(* Logix 5000 project; controller Joltek_RA_5069PLC002 vendor 1 type 14 code 226 rev 34.15; software revision 34.04 *)

TASK MainTask (continuous, watchdog 500 ms) : MainProgram
TASK SafetyTask (periodic, rate 20 ms, priority 10, watchdog 20 ms, safety) : SafetyProgram

MODULES
   Local : vendor 1 type 14 code 226 (5069 0, rev 34.15)
      Joltek_SW001 : vendor 1 type 12 code 231 (Ethernet 192.168.1.70, rev 13.8, Output RPI 1000 ms)
END_MODULES

TYPE UDT_ErrorDataLog :
STRUCT
   Time : UDT_Timestamp;
   DINTlog : DINT[10];
   REALlog : REAL[10];
END_STRUCT
END_TYPE

TYPE UDT_Line :
STRUCT
   Filler : UDT_Machine;
   Capper : UDT_Machine;
   Labeler : UDT_Machine;
   CasePAcker : UDT_Machine;
END_STRUCT
END_TYPE

TYPE UDT_Machine :
STRUCT
   Status : INT;
   Running : TIMER;
   Running_B : BOOL;
   CustomData : DINT[10];
   CustomREALData : REAL[10];
   Faulted : DINT;
END_STRUCT
END_TYPE

TYPE UDT_MachineData :
STRUCT
   CurrHourProdMade : INT;
   Prev120ShiftProdMade : INT[120];
   Last8HoursProdMade : INT[8];
   ResettableProdMade : DINT;
END_STRUCT
END_TYPE

TYPE UDT_Timestamp :
STRUCT
   Year : DINT;
   Month : DINT;
   Day : DINT;
   Hour : DINT;
   Minute : DINT;
   Second : DINT;
END_STRUCT
END_TYPE

TYPE UDT_TimestampedData :
STRUCT
   Hour : INT;
   Minute : INT;
   Second : INT;
   Data1 : DINT;
   Data2 : DINT;
   Data3 : DINT;
   Data_BOOL : BOOL[32];
   Data_REAL : REAL[5];
END_STRUCT
END_TYPE

VAR_GLOBAL   (* controller tags *)
   HMI_BOOL1 : BOOL[128] := ([0] := 1);
        [2]   // Filler - HMI | Station 1 Filling
        [3]   // Filler - HMI | Station 2 Filling
   HMI_INT : INT[100] := ([0] := 1, [1] := 96, [2] := 14, [3] := 16652, [4] := 88, [10] := 3, [11] := 40, [12] := 9134, [14] := 9, [20] := 2, [23] := 2056, [30] := 2, [31] := 9850, [32] := 70, [33] := 4100, [40] := 3, [41] := 9, [42] := 45, [50] := 4, [51] := 22, [52] := 7, [56] := 22, [57] := 7, [61] := 22, [62] := 7, [67] := 22, [68] := 7);
        [50].0   // Line - HIM | Start Permissive
        [3].13   // Filler HMI - Start Command
        [50].1   // Line - HIM | Start Command
        [50].2   // Line - HIM | Stop Permissive
        [50].3   // Line - HIM | Stop Command
        [23].1   // Labeler - Start Permissive
        [50].5   // Line - HIM | Fault Reset Command
        [23].3   // Labeler - Stop Permissive
        [23].4   // Labeler - HMI Stop Command
        [23].5   // Labeler - HMI Faulted Status
        [23].6   // Labeler - HMI Fault Reset Command
        [33].0   // Case Packer - HMI | Case Folding in Progress
        [33].1   // Case Packer - HMI | Case Gluing in Progress
        [33].10   // Case Packer - HMI | Start Permissive
        [33].11   // Case Packer - HMI | Start Command
        [33].12   // Case Packer - HMI | Stop Permissive
        [33].13   // Case Packer - HMI | Stop Command
        [33].15   // Case Packer - HMI | Clear Fault Command
        [41].0   // Palletizer - HMI | Currently Palletizing
        [14].6   // Capper - HMI | Fault Reset Command
        [41].1   // Palletizer - HMI | Start Permissive
        [23].2   // Labeler - HMI Start Command
        [23].0   // Labeler - Labeling in Process
        [3].12   // Filler - Start Permissive
        [41].2   // Palletizer - HMI | Start Command
        [14].2   // Capper - HMI | Start Command
        [41].7   // Palletizer - HMI | Clear Pallet Command
        [14].4   // Capper - HMI | Stop Command
        [4].2   // Filler - HMI | Add Bottles to Infeed
        [4].3   // Filler - HMI | Add Bottles to Infeed Permissive
        [4].4   // Overall - HMI | Count Reset Permissive
        [4].5   // Overall - HMI | Count Reset
        [4].7   // Overall - HMI | All Data Reset
        [4].6   // Overall - HMI | All Data Reset Permissive
   HMI_REAL : REAL[100] := ([0] := 46.01, [1] := 36.01, [2] := 100.0, [4] := 100.0, [7] := 100.0);
   LabelerNumberOfStops : COUNTER := (ACC := 16, DN := 1);
   LabelerStop_Data1ARR : DINT[100] := ([0] := 212, [1] := 209);
   LabelerStop_Data1CTR : CONTROL := (LEN := 100, POS := 2);
   LabelerStop_Data2CTR : CONTROL := (LEN := 100, POS := 5);
   LabelerStop_Hour : DINT := 10;
   LabelerStop_HourARR : DINT[100] := ([0] := 11, [1] := 11);
   LabelerStop_HourCTR : CONTROL := (LEN := 100, POS := 2);
   LabelerStop_MinCTR : CONTROL := (LEN := 100, POS := 2);
   LabelerStop_Minute : DINT := 2;
   LabelerStop_MinuteARR : DINT[100] := ([0] := 43, [1] := 43);
   LabelerStop_ONS : BOOL;
   LabelerStop_SecCTR : CONTROL := (LEN := 100, POS := 2);
   LabelerStop_Second : DINT := 37;
   LabelerStop_SecondARR : DINT[100] := ([0] := 11, [1] := 30);
   LabelerStopData : UDT_TimestampedData[100] := ([0].Hour := 12, [0].Minute := 24, [0].Second := 59, [0].Data1 := 193, [0].Data2 := 40, [0].Data3 := 6, [1].Hour := 12, [1].Minute := 25, [1].Second := 27, [1].Data1 := 188, [1].Data2 := 40, [1].Data3 := 5, [2].Hour := 22, [2].Minute := 24, [2].Second := 31, [2].Data1 := 188, [2].Data2 := 40, [2].Data3 := 5, [3].Hour := 10, [3].Second := 20, [3].Data1 := 249, [3].Data2 := 40, [3].Data3 := 2, [4].Hour := 10, [4].Minute := 2, [4].Second := 37, [4].Data1 := 246, [4].Data2 := 40, [4].Data3 := 5);
   LabelerStopDataONE : UDT_TimestampedData := (Hour := 10, Minute := 2, Second := 37, Data1 := 246, Data2 := 40, Data3 := 5);
   LabelerStops : COUNTER := (ACC := 3, CU := 1, DN := 1);
   Line1 : UDT_Line;
   Line34Pump3Motor342DischargeOfTank23_Sig : DINT;
   Line45Pump3MTR345InfeedRawIngredientFlou : DINT;
   Line6Pump1DischargeOfTank3 : DINT;
   Sys_DINT : DINT[100] := ([0] := 3, [1] := 1796, [2] := 6546, [3] := 49412, [4] := 96, [5] := 4601, [6] := 3601, [7] := 1, [8] := 1, [9] := 1, [10] := 1, [11] := 1, [12] := 1, [13] := 1, [14] := 1, [15] := 1, [16] := 1, [17] := 1, [18] := 1, [19] := 1, [20] := 1, [21] := 1, [22] := 1, [23] := 1, [24] := 1, [25] := 1, [26] := 1, [27] := 1, [28] := 1, [29] := 1, [30] := 1, [31] := 1, [32] := 1, [33] := 1, [34] := 1, [35] := 1, [36] := 1, [39] := 14, [40] := 52, [41] := 10000, [42] := 40, [43] := 9134, [44] := 516, [48] := 4, [49] := 9850, [51] := 205100, [53] := 70, [54] := 1, [55] := 20, [56] := 10000, [57] := 45, [58] := 22, [59] := 22, [60] := 7, [64] := 25, [65] := 22, [66] := 7);
        [0]   // Line 1 Motor 324 of the Conveyor 23 Discharge Pump 4-20mA Signal
        [40].4   // Capper - Start Capping Process
        [54].0   // Case Packer - Infeed Labeled Bottles Empty
        [1]   // Line 2 Motor 32334 of the Conveyor 2233 Discharge Pump 0-20mA Signal SCALED
        [55].1   // Palletizer - Stop
        [48].4   // Case Packer - Case Filling Station
        [3].4   // Filler - Alarm | Infeed Empty Bottle Conveyor Empty
        [48].5   // Case Packer - Gluing Station Case in Place
        [40].0   // Capper - Start
        [3].7   // Filler - Alarm | Discharge Filled Bottle Conveyor Almost Full
        [48].6   // Case Packer - Case Filled Ready
        [40].5   // Capper Discharge Conveyor Full
        [54].1   // Case Packer - Infeed Labeled Bottles Low
        [55].2   // Palletizer - Running
        [40].1   // Capper - Stop
        [3].6   // Filler - Alarm | Discharge Filled Bottle Conveyor Full
        [40].6   // Capper Discharge Conveyor Almost Full
        [40].2   // Capper - Running
        [3].2   // Filler - Running
        [44].0   // Labeler - Start
        [44].1   // Labeler - Stop
        [44].10   // Labeler - Unwind Station Almost Empty
        [44].2   // Labeler - Running
        [44].3   // Labeler - Faulted
        [44].5   // Labeler - Labeled Bottle Conveyor Full
        [44].6   // Labeler - Labeled Bottle Conveyor Almost Full
        [44].7   // Labeler - Capped Bottle Conveyor Empty
        [44].8   // Labeler - Capped Bottle Conveyor Almost Empty
        [44].9   // Labeler - Unwind Station Empty
        [46]   // Labeled Bollte Conveyor Count
        [48].0   // Case Packer - Start
        [48].7   // Case Packer - Gluing Station Case Start
        [3].3   // Filler - Faulted
        [55].3   // Palletizer - Faulted
        [54].2   // Case Packer - Cases Empty
        [54].3   // Case Packer - Cases Low
        [40].7   // Capper Infeed Conveyor Empty
        [3].5   // Filler - Alarm | Infeed Empty Bottle Conveyor Low
        [40].8   // Capper Infeed Conveyor Almost Empty
        [49]   // Case Packer - Empty Case Count
        [54].4   // Case Packer - Glue Tank Empty
        [43]   // Capper - Caps available in the hopper
        [55].4   // Palletizer - Case Placed by Robot
        [48].1   // Case Packer - Stop
        [4]   // Filler - Infeed Empty Bottle Count
        [48].2   // Case Packer - Running
        [51]   // Case Packer - Glue Station Level (10,000)
        [54].5   // Case Packer - Glue Tank Low
        [54].6   // Case Packer - Discharge Conveyor Full
        [48].3   // Case Packer - Faulted
        [54].7   // Case Packer - Discharge Conveyor Almost Full
        [40].3   // Capper - Faulted
        [3].1   // Filler - Stop
        [39]   // Filled Bottle Conveyor Count
        [3].12   // Test - Shift Change
        [3].0   // Filler - Start
        [3].8   // Filler - Bottle Filled
        [55].0   // Palletizer - Start
        [3].19   // Test - Hour Change
        [64]   // Current Hour of the Shift
        [65]   // Current Hour of the Shift
   Sys_FIFO_C : CONTROL[50] := ([0].LEN := 32, [0].POS := 32, [0].DN := 1, [1].LEN := 120, [1].EM := 1, [2].LEN := 120, [2].EM := 1, [3].LEN := 120, [3].EM := 1, [4].LEN := 120, [4].EM := 1, [5].LEN := 120, [5].EM := 1, [6].LEN := 120, [6].POS := 1, [7].DN := 1, [7].EM := 1, [8].DN := 1, [8].EM := 1, [9].DN := 1, [9].EM := 1, [10].DN := 1, [10].EM := 1);
   Sys_Timer : TIMER[100] := ([0].PRE := 50, [0].ACC := 39, [0].EN := 1, [0].TT := 1, [1].PRE := 150, [1].ACC := 139, [1].EN := 1, [1].TT := 1, [2].PRE := 2000, [2].ACC := 2000, [2].EN := 1, [2].DN := 1, [3].PRE := 200, [3].ACC := 18, [3].EN := 1, [3].TT := 1, [4].PRE := 200, [4].ACC := 18, [4].EN := 1, [4].TT := 1, [5].PRE := 1000000, [5].ACC := 8572, [5].EN := 1, [5].TT := 1, [10].PRE := 50, [10].ACC := 18, [10].EN := 1, [10].TT := 1, [11].PRE := 50, [12].PRE := 50, [13].PRE := 100, [14].PRE := 50, [14].ACC := 28, [14].EN := 1, [14].TT := 1);
   System_Date_Time : DINT[7] := ([0] := 2026, [1] := 1, [2] := 15, [3] := 23, [4] := 49, [5] := 38, [6] := 94001);
   Test_Bool : BOOL[64];
   TestBOOL : BOOL;
   TestControl : CONTROL;
   TestCounter : COUNTER;
   TestDINT : DINT;
   TestDINTArray : DINT[10];
   TestINT : INT;
   TestTimer : TIMER;
   TestTimerArr : TIMER[10];
END_VAR

PROGRAM MainProgram   (* main routine MainRoutine *)
VAR
   CapperData : UDT_MachineData := (CurrHourProdMade := 7, Prev120ShiftProdMade[2] := 449, Prev120ShiftProdMade[3] := 480, Prev120ShiftProdMade[4] := 480, Prev120ShiftProdMade[5] := 480, Prev120ShiftProdMade[6] := 480, Prev120ShiftProdMade[7] := 480, Prev120ShiftProdMade[8] := 480, Last8HoursProdMade[1] := 7);
   CasePackerData : UDT_MachineData;
   CurrentPos1 : DINT := 12;
   FillerData : UDT_MachineData := (CurrHourProdMade := 22, Prev120ShiftProdMade[2] := 226, Last8HoursProdMade[1] := 22);
   LabelerData : UDT_MachineData;
   PalletizerData : UDT_MachineData;
   shiftHour : INT := 1;
   Vlad_Test : BOOL[64] := ([0] := 1);
END_VAR

ROUTINE _01_System   (* ladder *)
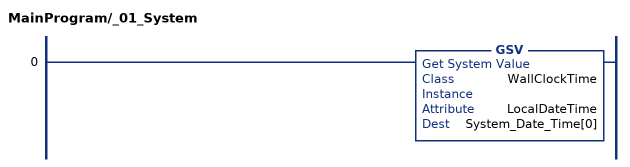
   0: GSV(WallClockTime,,LocalDateTime,System_Date_Time[0]);
END_ROUTINE

ROUTINE _02_Filler   (* ladder *)
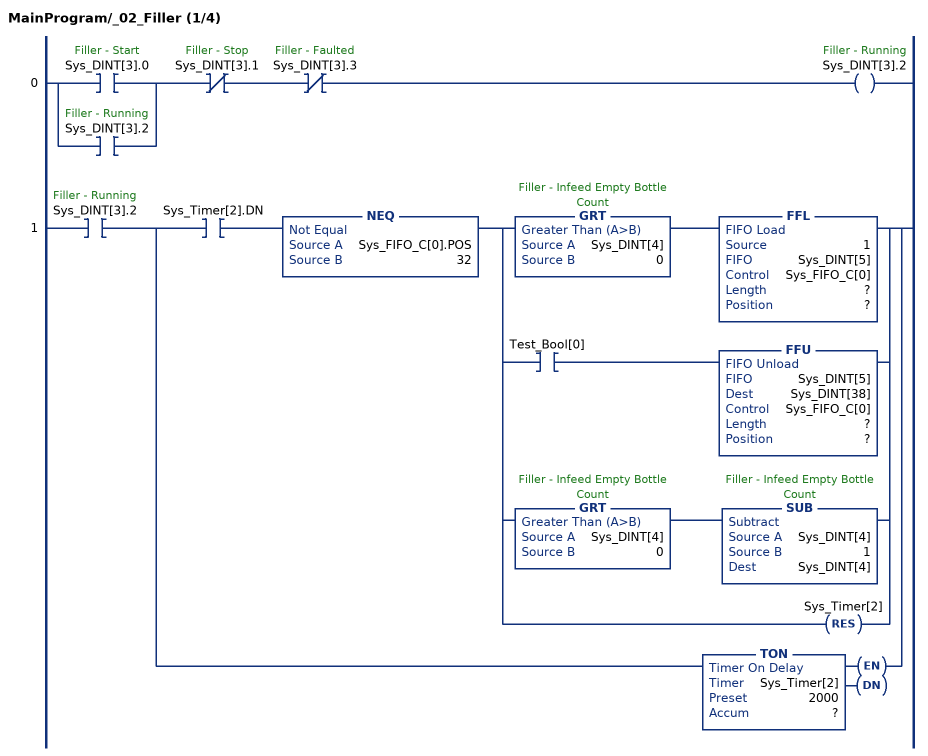
   0: [XIC(Sys_DINT[3].0) ,XIC(Sys_DINT[3].2) ]XIO(Sys_DINT[3].1)XIO(Sys_DINT[3].3)OTE(Sys_DINT[3].2);
   1: XIC(Sys_DINT[3].2)[XIC(Sys_Timer[2].DN) NEQ(Sys_FIFO_C[0].POS,32) [GRT(Sys_DINT[4],0) FFL(1,Sys_DINT[5],Sys_FIFO_C[0],?,?) ,XIC(Test_Bool[0]) FFU(Sys_DINT[5],Sys_DINT[38],Sys_FIFO_C[0],?,?) ,GRT(Sys_DINT[4],0) SUB(Sys_DINT[4],1,Sys_DINT[4]) ,RES(Sys_Timer[2]) ] ,TON(Sys_Timer[2],?,?) ];
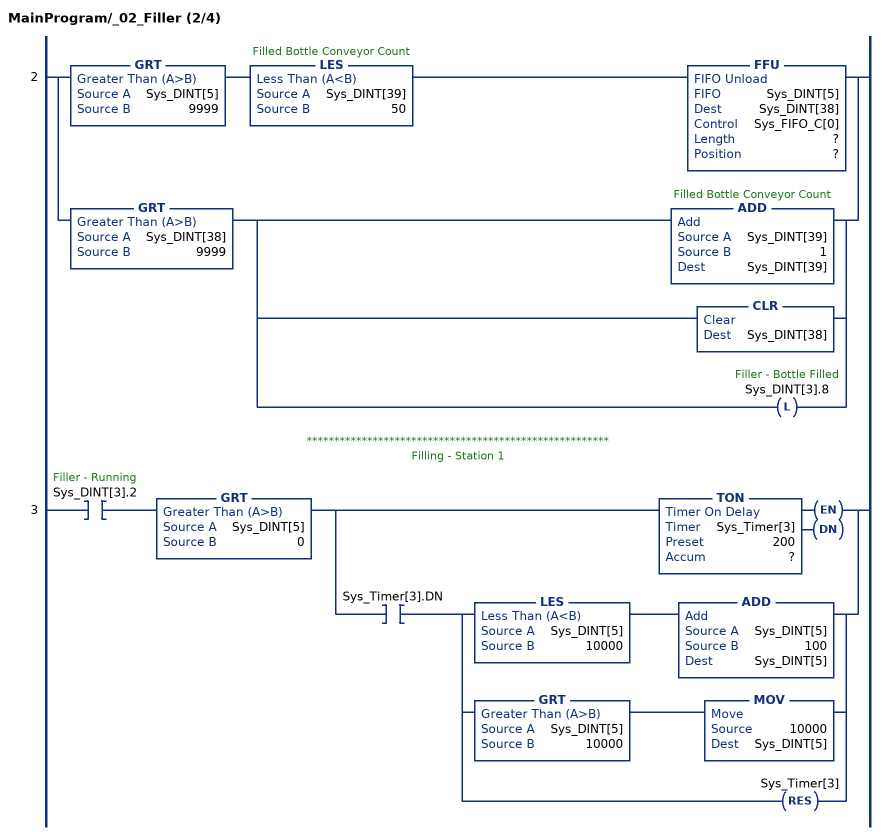
   2: [GRT(Sys_DINT[5],9999) LES(Sys_DINT[39],50) FFU(Sys_DINT[5],Sys_DINT[38],Sys_FIFO_C[0],?,?) ,GRT(Sys_DINT[38],9999) [ADD(Sys_DINT[39],1,Sys_DINT[39]) ,CLR(Sys_DINT[38]) ,OTL(Sys_DINT[3].8) ] ];
   // *******************************************************
   // Filling - Station 1
   3: XIC(Sys_DINT[3].2)GRT(Sys_DINT[5],0)[TON(Sys_Timer[3],?,?) ,XIC(Sys_Timer[3].DN) [LES(Sys_DINT[5],10000) ADD(Sys_DINT[5],100,Sys_DINT[5]) ,GRT(Sys_DINT[5],10000) MOV(10000,Sys_DINT[5]) ,RES(Sys_Timer[3]) ] ];
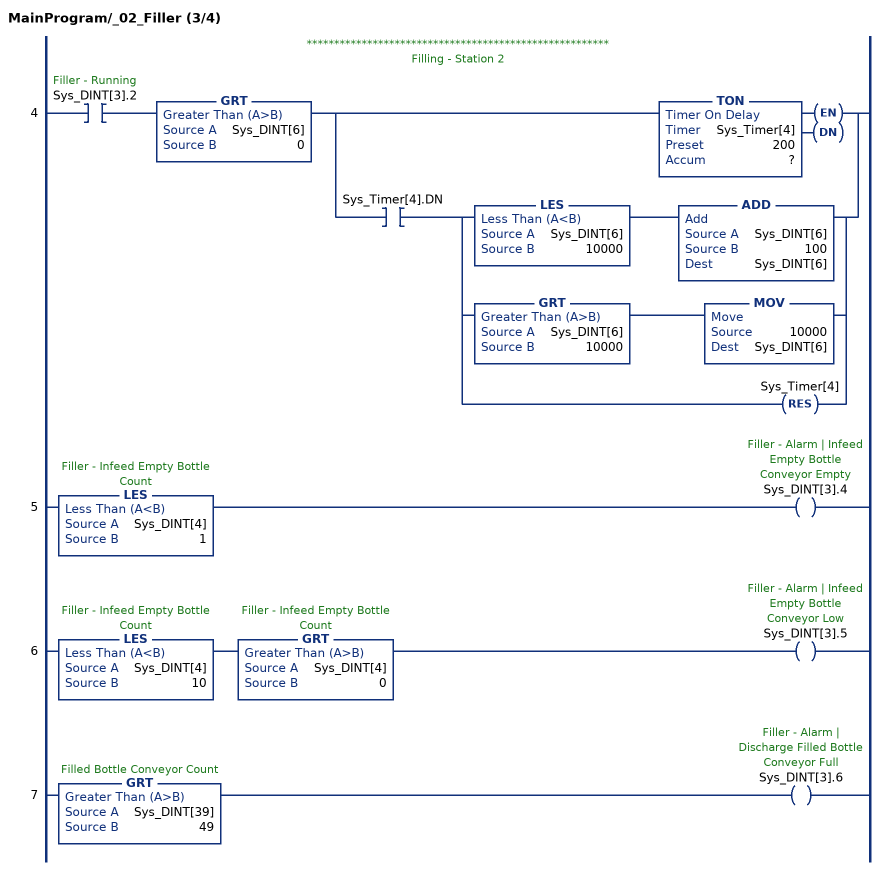
   // *******************************************************
   // Filling - Station 2
   4: XIC(Sys_DINT[3].2)GRT(Sys_DINT[6],0)[TON(Sys_Timer[4],?,?) ,XIC(Sys_Timer[4].DN) [LES(Sys_DINT[6],10000) ADD(Sys_DINT[6],100,Sys_DINT[6]) ,GRT(Sys_DINT[6],10000) MOV(10000,Sys_DINT[6]) ,RES(Sys_Timer[4]) ] ];
   5: LES(Sys_DINT[4],1)OTE(Sys_DINT[3].4);
   6: LES(Sys_DINT[4],10)GRT(Sys_DINT[4],0)OTE(Sys_DINT[3].5);
   7: GRT(Sys_DINT[39],49)OTE(Sys_DINT[3].6);
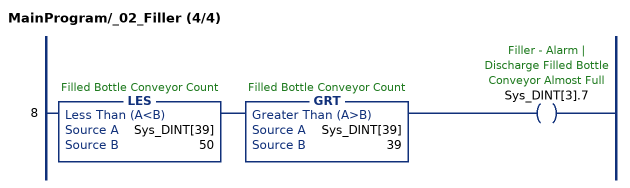
   8: LES(Sys_DINT[39],50)GRT(Sys_DINT[39],39)OTE(Sys_DINT[3].7);
END_ROUTINE

ROUTINE _03_Capper   (* ladder *)
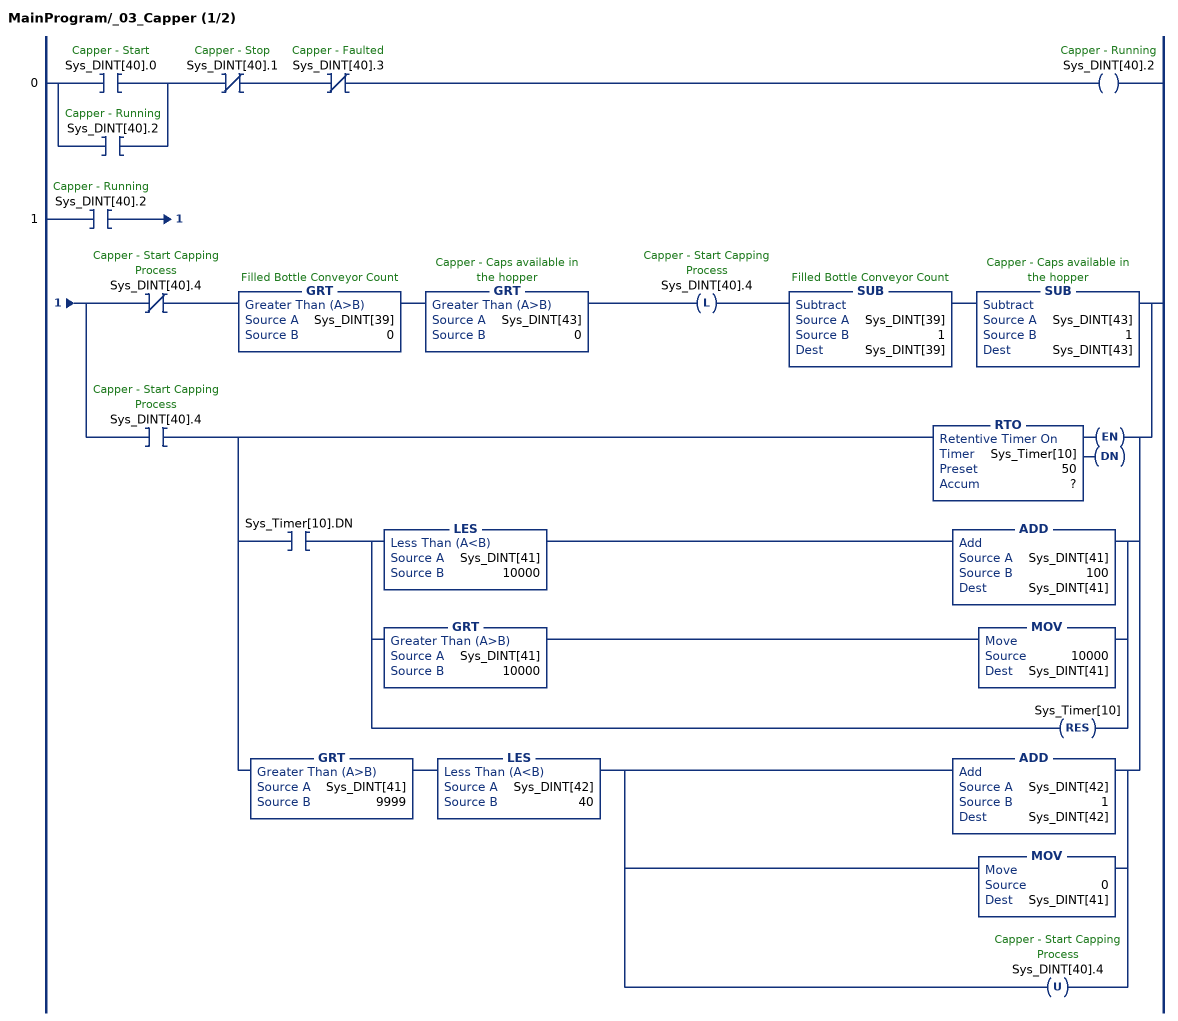
   0: [XIC(Sys_DINT[40].0) ,XIC(Sys_DINT[40].2) ]XIO(Sys_DINT[40].1)XIO(Sys_DINT[40].3)OTE(Sys_DINT[40].2);
   1: XIC(Sys_DINT[40].2)[XIO(Sys_DINT[40].4) GRT(Sys_DINT[39],0) GRT(Sys_DINT[43],0) OTL(Sys_DINT[40].4) SUB(Sys_DINT[39],1,Sys_DINT[39]) SUB(Sys_DINT[43],1,Sys_DINT[43]) ,XIC(Sys_DINT[40].4) [RTO(Sys_Timer[10],?,?) ,XIC(Sys_Timer[10].DN) [LES(Sys_DINT[41],10000) ADD(Sys_DINT[41],100,Sys_DINT[41]) ,GRT(Sys_DINT[41],10000) MOV(10000,Sys_DINT[41]) ,RES(Sys_Timer[10]) ] ,GRT(Sys_DINT[41],9999) LES(Sys_DINT[42],40) [ADD(Sys_DINT[42],1,Sys_DINT[42]) ,MOV(0,Sys_DINT[41]) ,OTU(Sys_DINT[40].4) ] ] ];
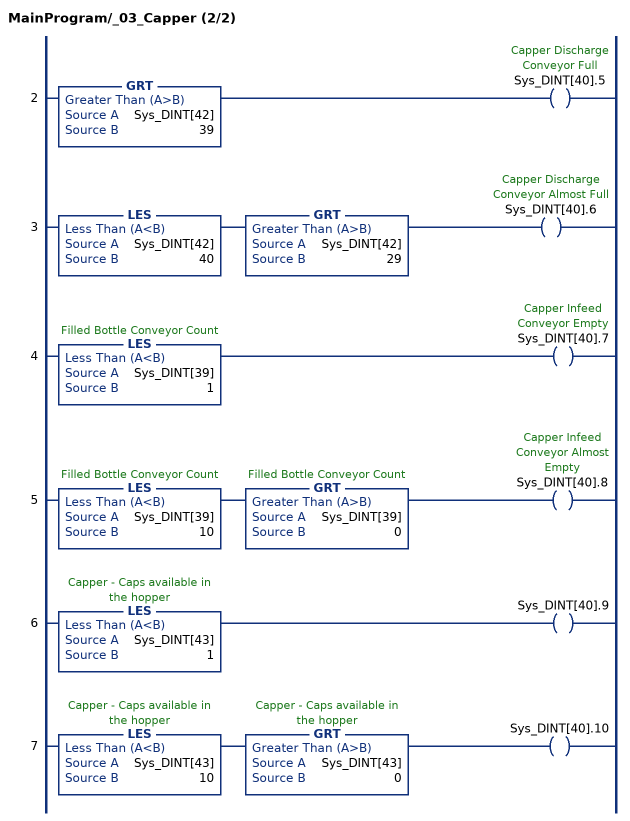
   2: GRT(Sys_DINT[42],39)OTE(Sys_DINT[40].5);
   3: LES(Sys_DINT[42],40)GRT(Sys_DINT[42],29)OTE(Sys_DINT[40].6);
   4: LES(Sys_DINT[39],1)OTE(Sys_DINT[40].7);
   5: LES(Sys_DINT[39],10)GRT(Sys_DINT[39],0)OTE(Sys_DINT[40].8);
   6: LES(Sys_DINT[43],1)OTE(Sys_DINT[40].9);
   7: LES(Sys_DINT[43],10)GRT(Sys_DINT[43],0)OTE(Sys_DINT[40].10);
END_ROUTINE

ROUTINE _04_Labeler   (* ladder *)
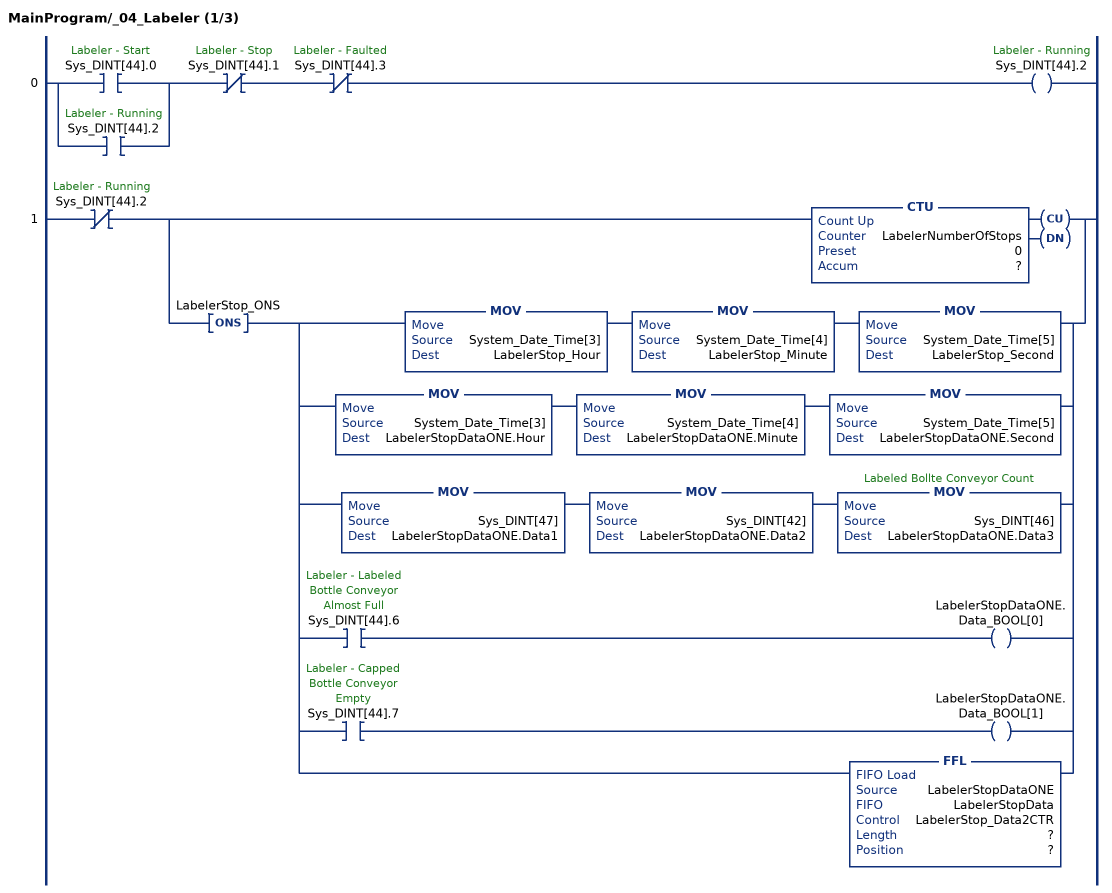
   0: [XIC(Sys_DINT[44].0) ,XIC(Sys_DINT[44].2) ]XIO(Sys_DINT[44].1)XIO(Sys_DINT[44].3)OTE(Sys_DINT[44].2);
   1: XIO(Sys_DINT[44].2)[CTU(LabelerNumberOfStops,?,?) ,ONS(LabelerStop_ONS) [MOV(System_Date_Time[3],LabelerStop_Hour) MOV(System_Date_Time[4],LabelerStop_Minute) MOV(System_Date_Time[5],LabelerStop_Second) ,[MOV(System_Date_Time[3],LabelerStopDataONE.Hour) MOV(System_Date_Time[4],LabelerStopDataONE.Minute) MOV(System_Date_Time[5],LabelerStopDataONE.Second) ,MOV(Sys_DINT[47],LabelerStopDataONE.Data1) MOV(Sys_DINT[42],LabelerStopDataONE.Data2) MOV(Sys_DINT[46],LabelerStopDataONE.Data3) ,[XIC(Sys_DINT[44].6) OTE(LabelerStopDataONE.Data_BOOL[0]) ,XIC(Sys_DINT[44].7) OTE(LabelerStopDataONE.Data_BOOL[1]) ] ,FFL(LabelerStopDataONE,LabelerStopData,LabelerStop_Data2CTR,?,?) ] ] ];
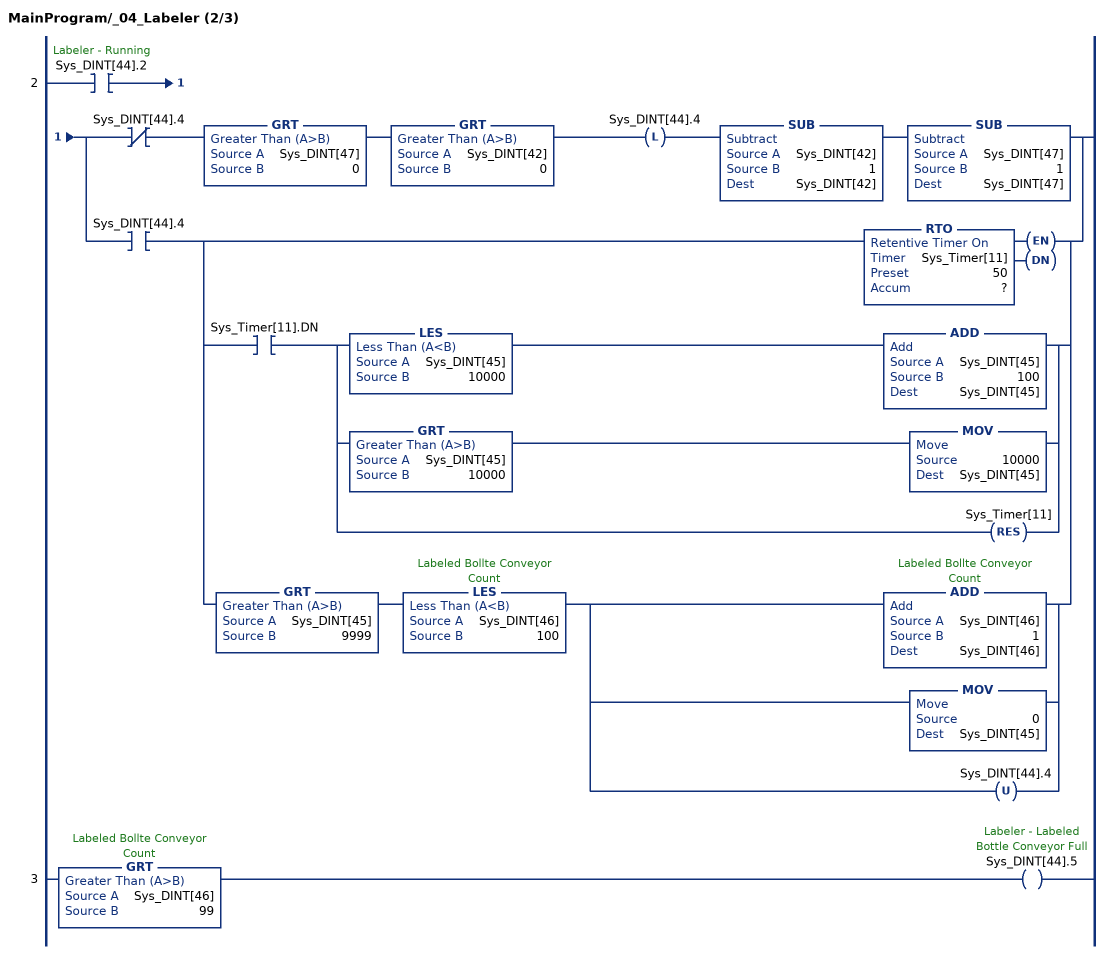
   2: XIC(Sys_DINT[44].2)[XIO(Sys_DINT[44].4) GRT(Sys_DINT[47],0) GRT(Sys_DINT[42],0) OTL(Sys_DINT[44].4) SUB(Sys_DINT[42],1,Sys_DINT[42]) SUB(Sys_DINT[47],1,Sys_DINT[47]) ,XIC(Sys_DINT[44].4) [RTO(Sys_Timer[11],?,?) ,XIC(Sys_Timer[11].DN) [LES(Sys_DINT[45],10000) ADD(Sys_DINT[45],100,Sys_DINT[45]) ,GRT(Sys_DINT[45],10000) MOV(10000,Sys_DINT[45]) ,RES(Sys_Timer[11]) ] ,GRT(Sys_DINT[45],9999) LES(Sys_DINT[46],100) [ADD(Sys_DINT[46],1,Sys_DINT[46]) ,MOV(0,Sys_DINT[45]) ,OTU(Sys_DINT[44].4) ] ] ];
   3: GRT(Sys_DINT[46],99)OTE(Sys_DINT[44].5);
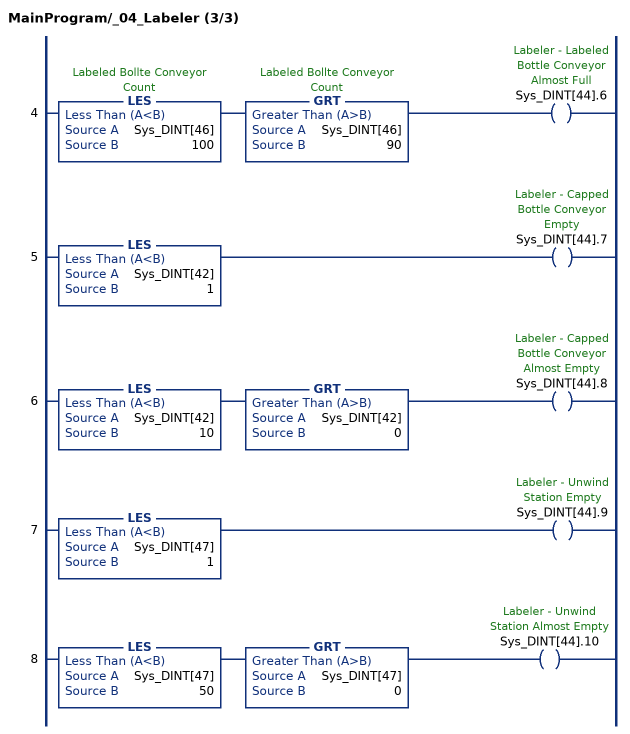
   4: LES(Sys_DINT[46],100)GRT(Sys_DINT[46],90)OTE(Sys_DINT[44].6);
   5: LES(Sys_DINT[42],1)OTE(Sys_DINT[44].7);
   6: LES(Sys_DINT[42],10)GRT(Sys_DINT[42],0)OTE(Sys_DINT[44].8);
   7: LES(Sys_DINT[47],1)OTE(Sys_DINT[44].9);
   8: LES(Sys_DINT[47],50)GRT(Sys_DINT[47],0)OTE(Sys_DINT[44].10);
END_ROUTINE

ROUTINE _05_CasePacker   (* ladder *)
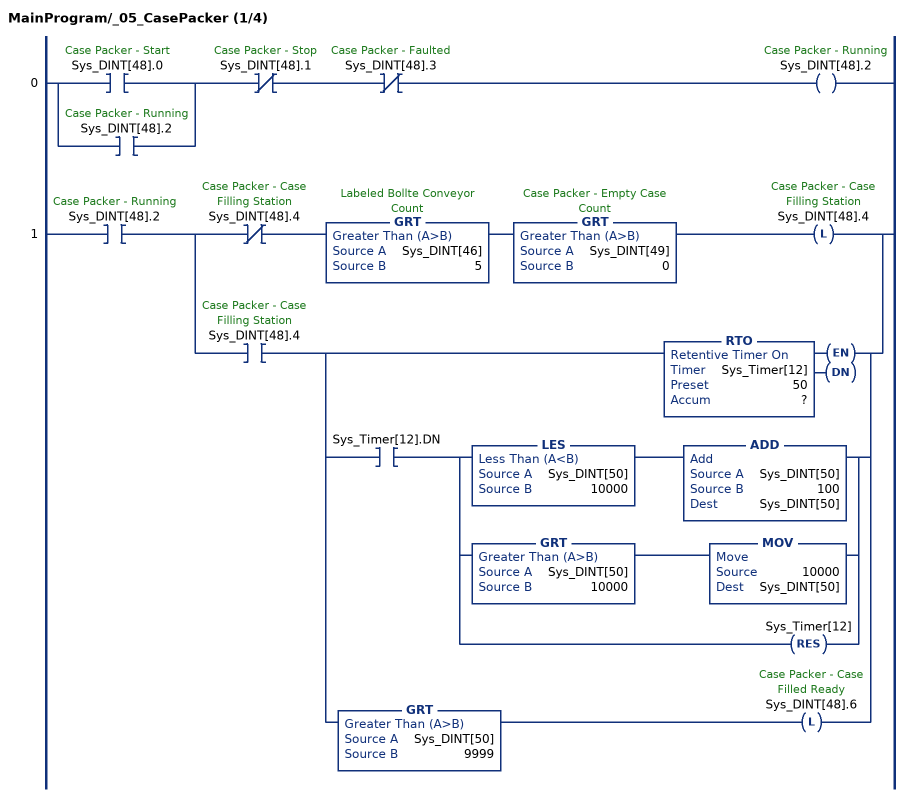
   0: [XIC(Sys_DINT[48].0) ,XIC(Sys_DINT[48].2) ]XIO(Sys_DINT[48].1)XIO(Sys_DINT[48].3)OTE(Sys_DINT[48].2);
   1: XIC(Sys_DINT[48].2)[XIO(Sys_DINT[48].4) GRT(Sys_DINT[46],5) GRT(Sys_DINT[49],0) OTL(Sys_DINT[48].4) ,XIC(Sys_DINT[48].4) [RTO(Sys_Timer[12],?,?) ,XIC(Sys_Timer[12].DN) [LES(Sys_DINT[50],10000) ADD(Sys_DINT[50],100,Sys_DINT[50]) ,GRT(Sys_DINT[50],10000) MOV(10000,Sys_DINT[50]) ,RES(Sys_Timer[12]) ] ,GRT(Sys_DINT[50],9999) OTL(Sys_DINT[48].6) ] ];
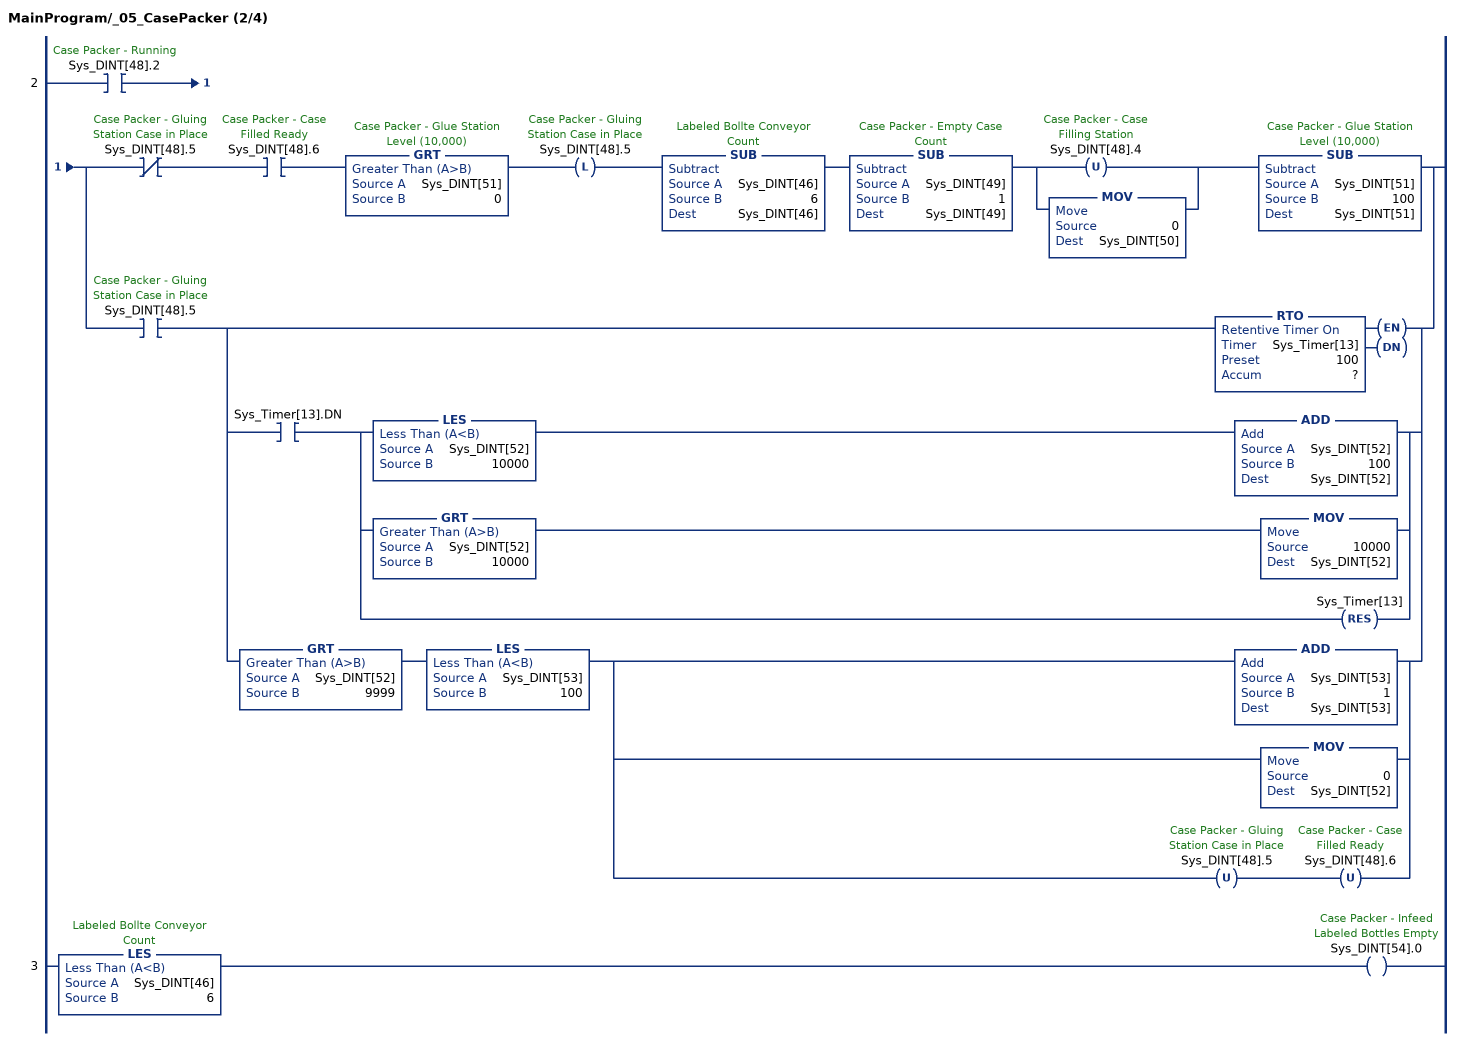
   2: XIC(Sys_DINT[48].2)[XIO(Sys_DINT[48].5) XIC(Sys_DINT[48].6) GRT(Sys_DINT[51],0) OTL(Sys_DINT[48].5) SUB(Sys_DINT[46],6,Sys_DINT[46]) SUB(Sys_DINT[49],1,Sys_DINT[49]) [OTU(Sys_DINT[48].4) ,MOV(0,Sys_DINT[50]) ] SUB(Sys_DINT[51],100,Sys_DINT[51]) ,XIC(Sys_DINT[48].5) [RTO(Sys_Timer[13],?,?) ,XIC(Sys_Timer[13].DN) [LES(Sys_DINT[52],10000) ADD(Sys_DINT[52],100,Sys_DINT[52]) ,GRT(Sys_DINT[52],10000) MOV(10000,Sys_DINT[52]) ,RES(Sys_Timer[13]) ] ,GRT(Sys_DINT[52],9999) LES(Sys_DINT[53],100) [ADD(Sys_DINT[53],1,Sys_DINT[53]) ,MOV(0,Sys_DINT[52]) ,OTU(Sys_DINT[48].5) OTU(Sys_DINT[48].6) ] ] ];
   3: LES(Sys_DINT[46],6)OTE(Sys_DINT[54].0);
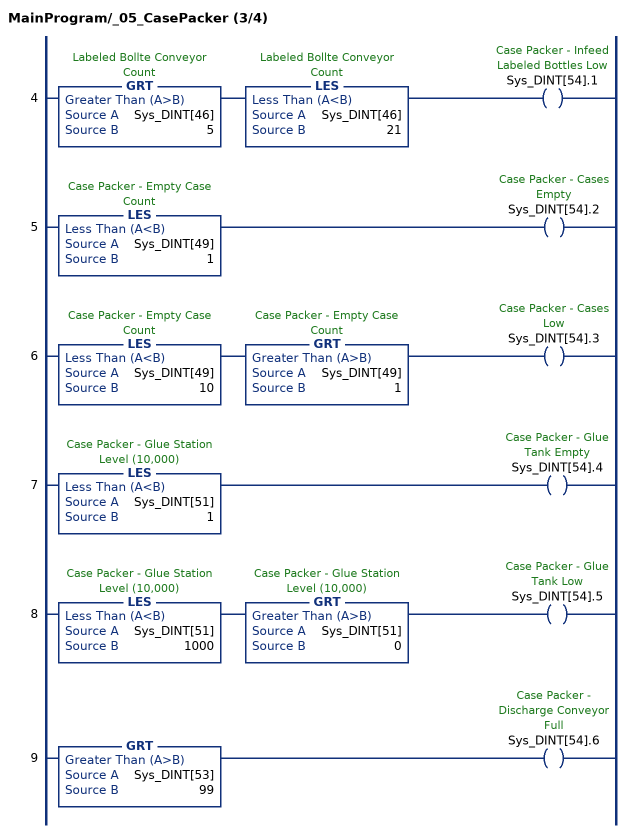
   4: GRT(Sys_DINT[46],5)LES(Sys_DINT[46],21)OTE(Sys_DINT[54].1);
   5: LES(Sys_DINT[49],1)OTE(Sys_DINT[54].2);
   6: LES(Sys_DINT[49],10)GRT(Sys_DINT[49],1)OTE(Sys_DINT[54].3);
   7: LES(Sys_DINT[51],1)OTE(Sys_DINT[54].4);
   8: LES(Sys_DINT[51],1000)GRT(Sys_DINT[51],0)OTE(Sys_DINT[54].5);
   9: GRT(Sys_DINT[53],99)OTE(Sys_DINT[54].6);
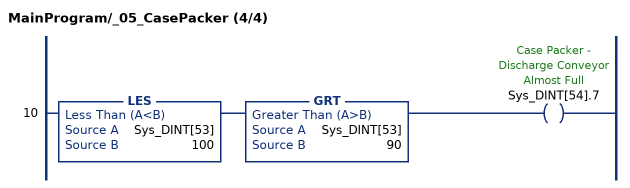
   10: LES(Sys_DINT[53],100)GRT(Sys_DINT[53],90)OTE(Sys_DINT[54].7);
END_ROUTINE

ROUTINE _06_Palletizer   (* ladder *)
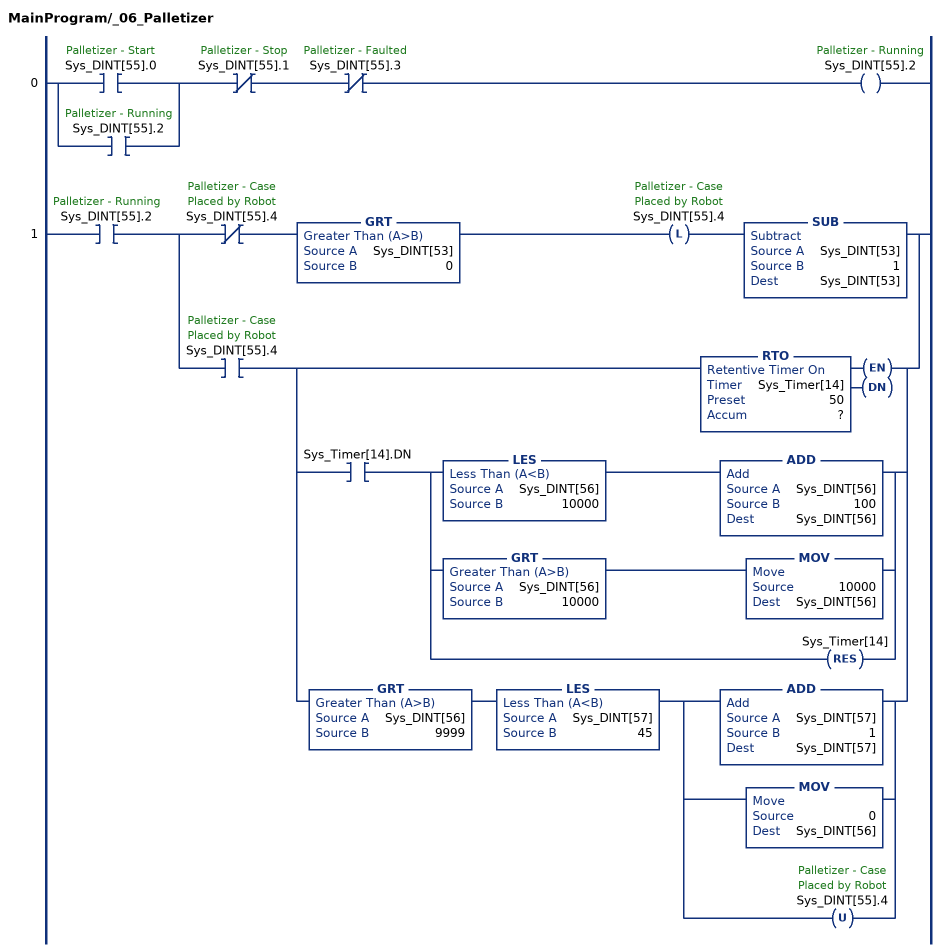
   0: [XIC(Sys_DINT[55].0) ,XIC(Sys_DINT[55].2) ]XIO(Sys_DINT[55].1)XIO(Sys_DINT[55].3)OTE(Sys_DINT[55].2);
   1: XIC(Sys_DINT[55].2)[XIO(Sys_DINT[55].4) GRT(Sys_DINT[53],0) OTL(Sys_DINT[55].4) SUB(Sys_DINT[53],1,Sys_DINT[53]) ,XIC(Sys_DINT[55].4) [RTO(Sys_Timer[14],?,?) ,XIC(Sys_Timer[14].DN) [LES(Sys_DINT[56],10000) ADD(Sys_DINT[56],100,Sys_DINT[56]) ,GRT(Sys_DINT[56],10000) MOV(10000,Sys_DINT[56]) ,RES(Sys_Timer[14]) ] ,GRT(Sys_DINT[56],9999) LES(Sys_DINT[57],45) [ADD(Sys_DINT[57],1,Sys_DINT[57]) ,MOV(0,Sys_DINT[56]) ,OTU(Sys_DINT[55].4) ] ] ];
END_ROUTINE

ROUTINE _50_HMI_Interface   (* ladder *)
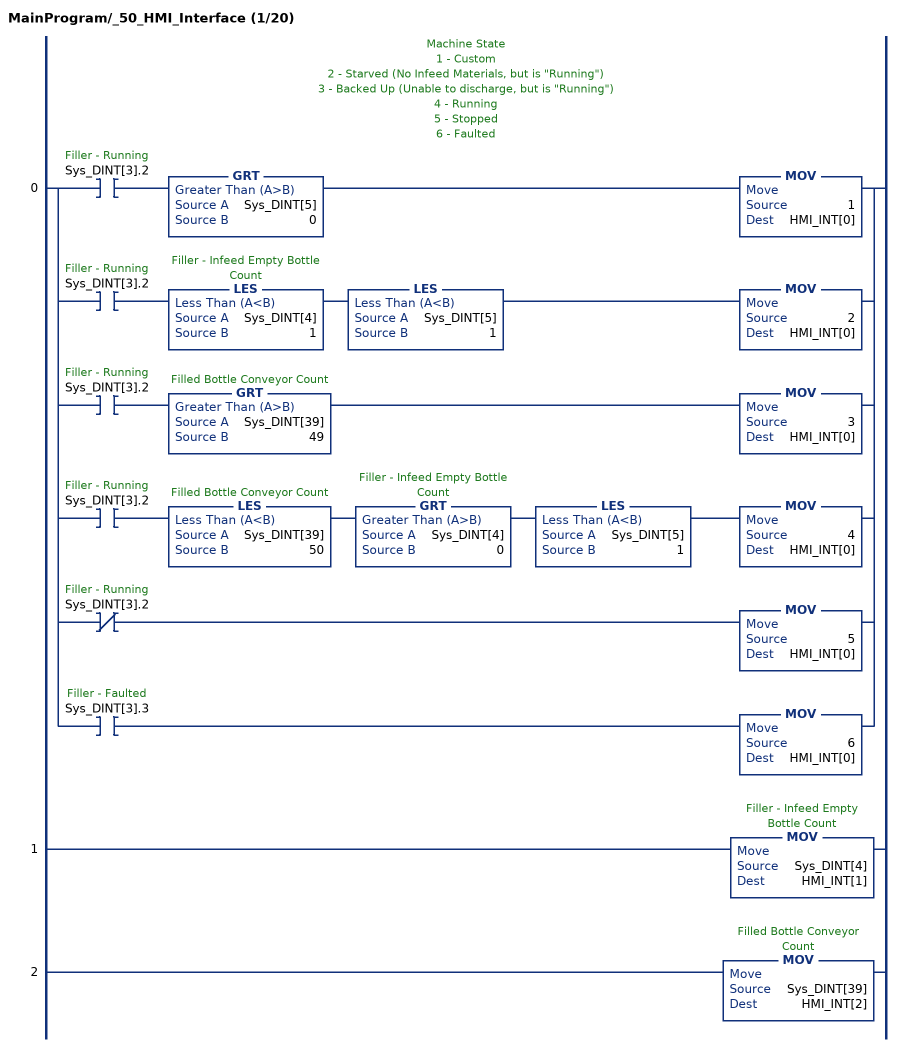
   // Machine State
   // 1 - Custom
   // 2 - Starved (No Infeed Materials, but is "Running")
   // 3 - Backed Up (Unable to discharge, but is "Running")
   // 4 - Running
   // 5 - Stopped
   // 6 - Faulted
   0: [XIC(Sys_DINT[3].2) GRT(Sys_DINT[5],0) MOV(1,HMI_INT[0]) ,XIC(Sys_DINT[3].2) LES(Sys_DINT[4],1) LES(Sys_DINT[5],1) MOV(2,HMI_INT[0]) ,XIC(Sys_DINT[3].2) GRT(Sys_DINT[39],49) MOV(3,HMI_INT[0]) ,XIC(Sys_DINT[3].2) LES(Sys_DINT[39],50) GRT(Sys_DINT[4],0) LES(Sys_DINT[5],1) MOV(4,HMI_INT[0]) ,XIO(Sys_DINT[3].2) MOV(5,HMI_INT[0]) ,XIC(Sys_DINT[3].3) MOV(6,HMI_INT[0]) ];
   1: MOV(Sys_DINT[4],HMI_INT[1]);
   2: MOV(Sys_DINT[39],HMI_INT[2]);
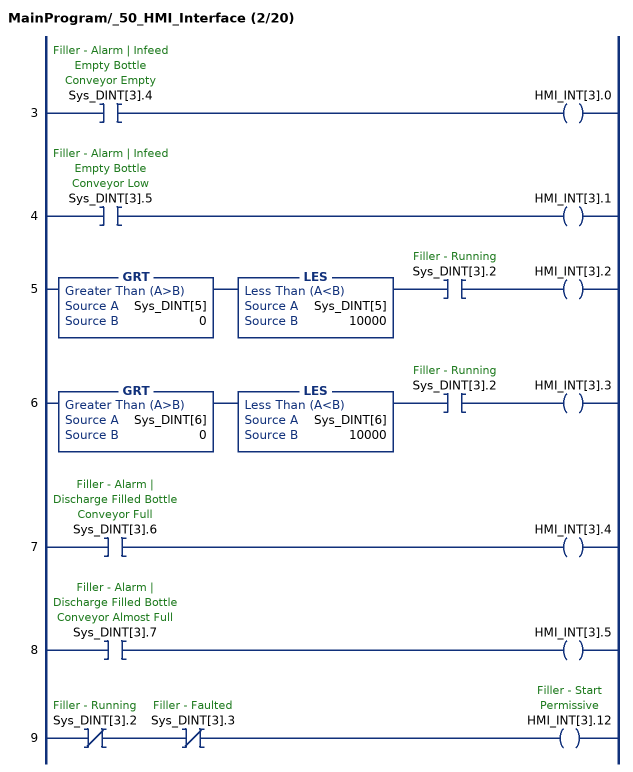
   3: XIC(Sys_DINT[3].4)OTE(HMI_INT[3].0);
   4: XIC(Sys_DINT[3].5)OTE(HMI_INT[3].1);
   5: GRT(Sys_DINT[5],0)LES(Sys_DINT[5],10000)XIC(Sys_DINT[3].2)OTE(HMI_INT[3].2);
   6: GRT(Sys_DINT[6],0)LES(Sys_DINT[6],10000)XIC(Sys_DINT[3].2)OTE(HMI_INT[3].3);
   7: XIC(Sys_DINT[3].6)OTE(HMI_INT[3].4);
   8: XIC(Sys_DINT[3].7)OTE(HMI_INT[3].5);
   9: XIO(Sys_DINT[3].2)XIO(Sys_DINT[3].3)OTE(HMI_INT[3].12);
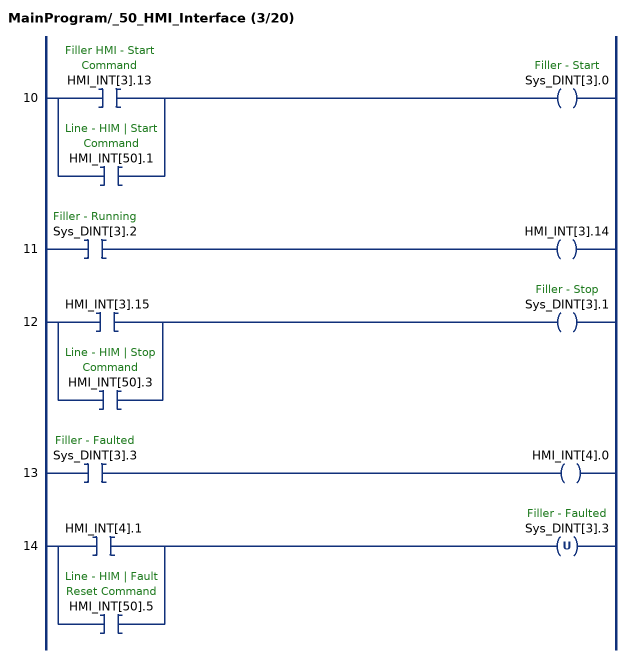
   10: [XIC(HMI_INT[3].13) ,XIC(HMI_INT[50].1) ]OTE(Sys_DINT[3].0);
   11: XIC(Sys_DINT[3].2)OTE(HMI_INT[3].14);
   12: [XIC(HMI_INT[3].15) ,XIC(HMI_INT[50].3) ]OTE(Sys_DINT[3].1);
   13: XIC(Sys_DINT[3].3)OTE(HMI_INT[4].0);
   14: [XIC(HMI_INT[4].1) ,XIC(HMI_INT[50].5) ]OTU(Sys_DINT[3].3);
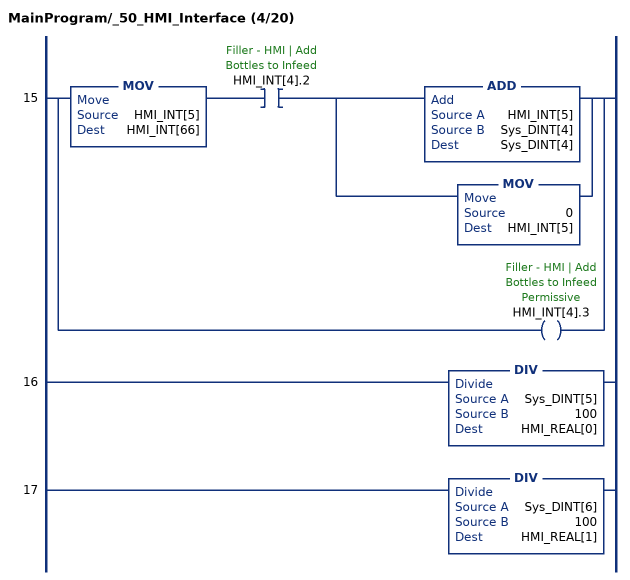
   15: [MOV(HMI_INT[5],HMI_INT[66]) XIC(HMI_INT[4].2) [ADD(HMI_INT[5],Sys_DINT[4],Sys_DINT[4]) ,MOV(0,HMI_INT[5]) ] ,OTE(HMI_INT[4].3) ];
   16: DIV(Sys_DINT[5],100,HMI_REAL[0]);
   17: DIV(Sys_DINT[6],100,HMI_REAL[1]);
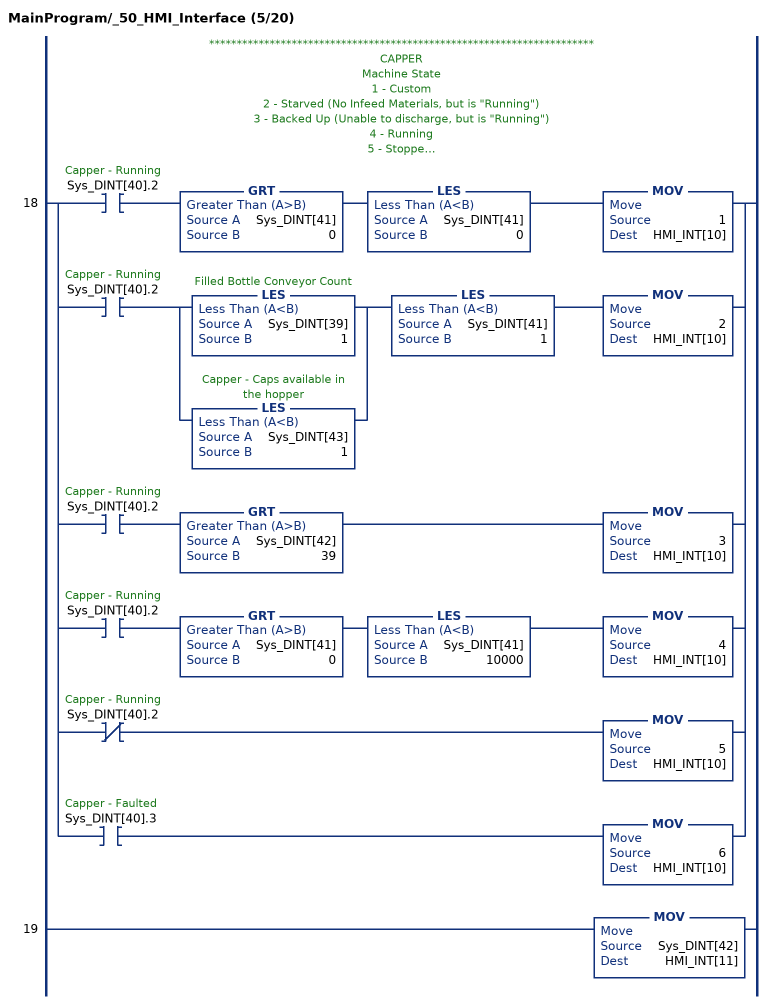
   // **********************************************************************
   // CAPPER
   // Machine State
   // 1 - Custom
   // 2 - Starved (No Infeed Materials, but is "Running")
   // 3 - Backed Up (Unable to discharge, but is "Running")
   // 4 - Running
   // 5 - Stopped
   // 6 - Faulted
   18: [XIC(Sys_DINT[40].2) GRT(Sys_DINT[41],0) LES(Sys_DINT[41],0) MOV(1,HMI_INT[10]) ,XIC(Sys_DINT[40].2) [LES(Sys_DINT[39],1) ,LES(Sys_DINT[43],1) ] LES(Sys_DINT[41],1) MOV(2,HMI_INT[10]) ,XIC(Sys_DINT[40].2) GRT(Sys_DINT[42],39) MOV(3,HMI_INT[10]) ,XIC(Sys_DINT[40].2) GRT(Sys_DINT[41],0) LES(Sys_DINT[41],10000) MOV(4,HMI_INT[10]) ,XIO(Sys_DINT[40].2) MOV(5,HMI_INT[10]) ,XIC(Sys_DINT[40].3) MOV(6,HMI_INT[10]) ];
   19: MOV(Sys_DINT[42],HMI_INT[11]);
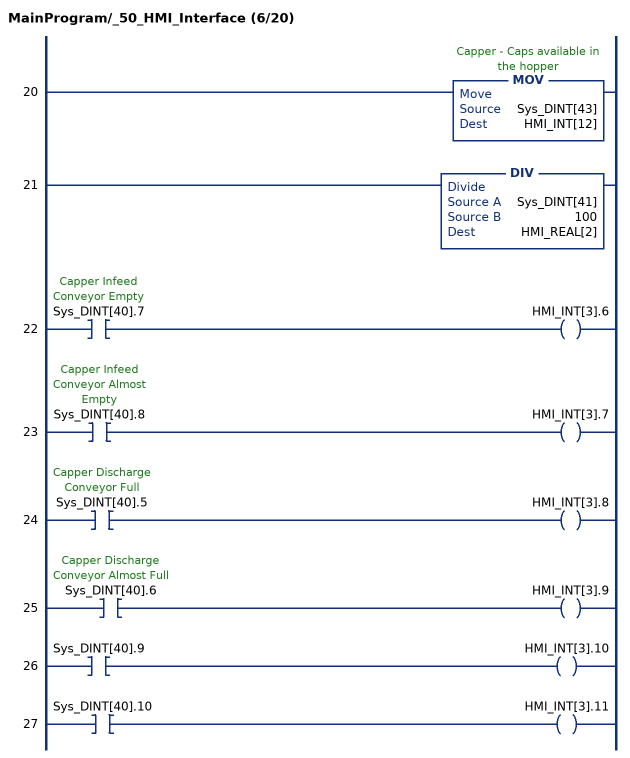
   20: MOV(Sys_DINT[43],HMI_INT[12]);
   21: DIV(Sys_DINT[41],100,HMI_REAL[2]);
   22: XIC(Sys_DINT[40].7)OTE(HMI_INT[3].6);
   23: XIC(Sys_DINT[40].8)OTE(HMI_INT[3].7);
   24: XIC(Sys_DINT[40].5)OTE(HMI_INT[3].8);
   25: XIC(Sys_DINT[40].6)OTE(HMI_INT[3].9);
   26: XIC(Sys_DINT[40].9)OTE(HMI_INT[3].10);
   27: XIC(Sys_DINT[40].10)OTE(HMI_INT[3].11);
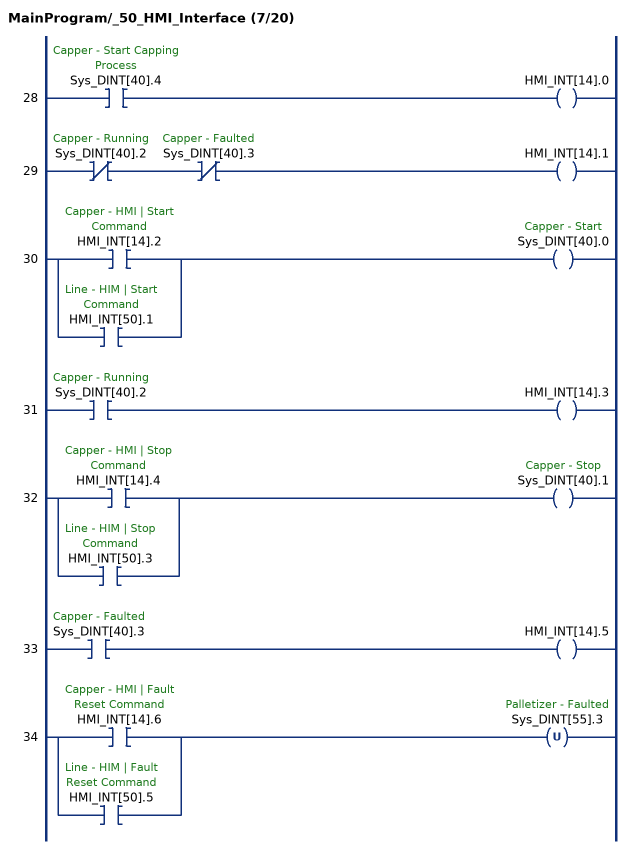
   28: XIC(Sys_DINT[40].4)OTE(HMI_INT[14].0);
   29: XIO(Sys_DINT[40].2)XIO(Sys_DINT[40].3)OTE(HMI_INT[14].1);
   30: [XIC(HMI_INT[14].2) ,XIC(HMI_INT[50].1) ]OTE(Sys_DINT[40].0);
   31: XIC(Sys_DINT[40].2)OTE(HMI_INT[14].3);
   32: [XIC(HMI_INT[14].4) ,XIC(HMI_INT[50].3) ]OTE(Sys_DINT[40].1);
   33: XIC(Sys_DINT[40].3)OTE(HMI_INT[14].5);
   34: [XIC(HMI_INT[14].6) ,XIC(HMI_INT[50].5) ]OTU(Sys_DINT[55].3);
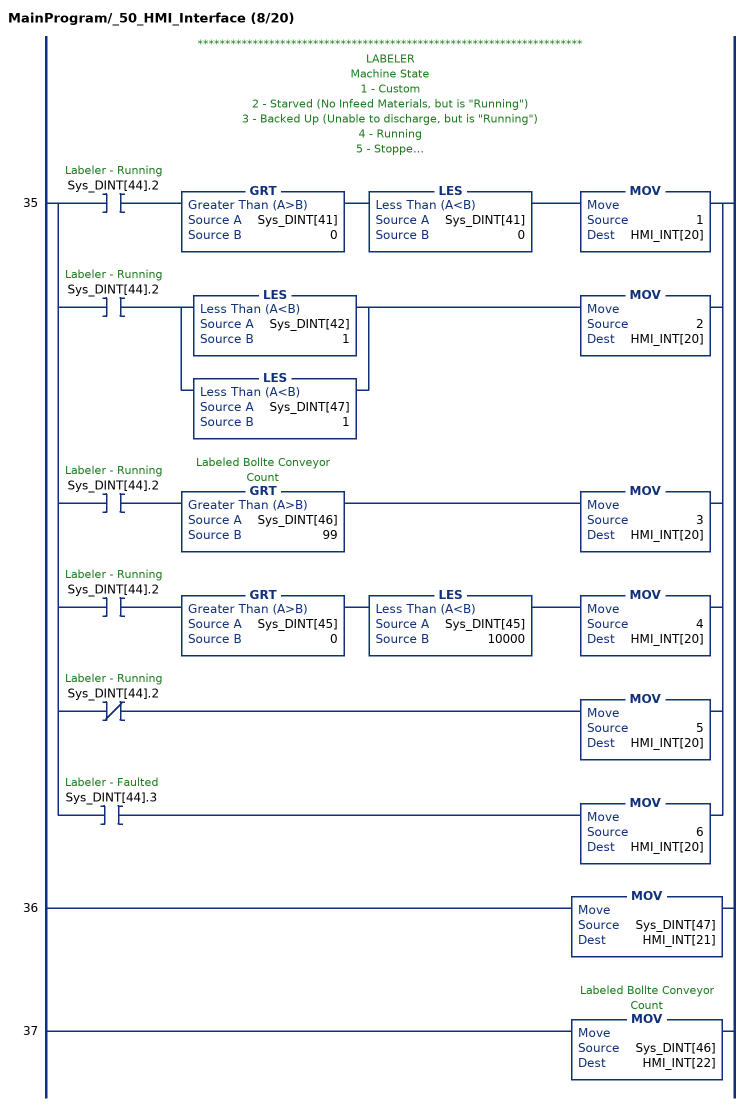
   // **********************************************************************
   // LABELER
   // Machine State
   // 1 - Custom
   // 2 - Starved (No Infeed Materials, but is "Running")
   // 3 - Backed Up (Unable to discharge, but is "Running")
   // 4 - Running
   // 5 - Stopped
   // 6 - Faulted
   35: [XIC(Sys_DINT[44].2) GRT(Sys_DINT[41],0) LES(Sys_DINT[41],0) MOV(1,HMI_INT[20]) ,XIC(Sys_DINT[44].2) [LES(Sys_DINT[42],1) ,LES(Sys_DINT[47],1) ] MOV(2,HMI_INT[20]) ,XIC(Sys_DINT[44].2) GRT(Sys_DINT[46],99) MOV(3,HMI_INT[20]) ,XIC(Sys_DINT[44].2) GRT(Sys_DINT[45],0) LES(Sys_DINT[45],10000) MOV(4,HMI_INT[20]) ,XIO(Sys_DINT[44].2) MOV(5,HMI_INT[20]) ,XIC(Sys_DINT[44].3) MOV(6,HMI_INT[20]) ];
   36: MOV(Sys_DINT[47],HMI_INT[21]);
   37: MOV(Sys_DINT[46],HMI_INT[22]);
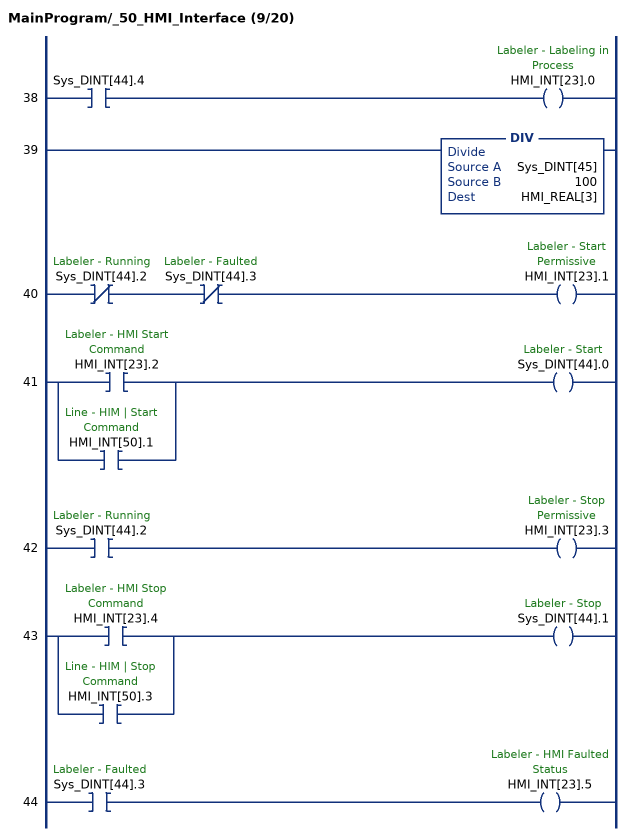
   38: XIC(Sys_DINT[44].4)OTE(HMI_INT[23].0);
   39: DIV(Sys_DINT[45],100,HMI_REAL[3]);
   40: XIO(Sys_DINT[44].2)XIO(Sys_DINT[44].3)OTE(HMI_INT[23].1);
   41: [XIC(HMI_INT[23].2) ,XIC(HMI_INT[50].1) ]OTE(Sys_DINT[44].0);
   42: XIC(Sys_DINT[44].2)OTE(HMI_INT[23].3);
   43: [XIC(HMI_INT[23].4) ,XIC(HMI_INT[50].3) ]OTE(Sys_DINT[44].1);
   44: XIC(Sys_DINT[44].3)OTE(HMI_INT[23].5);
